(* PLC project BE_Framework BA.project, CODESYS CODESYS V3.5 SP13 Patch 2 *)
(* stored: creationDateTime 2018-12-11T11:00:35.04202, modificationDateTime 2018-12-11T11:00:22.0036737 *)

PROGRAM LB01_FF1_Analog_ST
VAR
	local:strFan_Analog;
	localGP:strSensor2_Regulator;
	ControlFan: _BE_Fan;
	FbRegulator: _BE_Regulator;
	_BE_Fan2: _BE_Fan_2;
	reset_en: RS;
	AlarmFbAl03: _BE_AlarmAckRequired;
	AlarmFbAl02: _BE_AlarmAckRequired;
	fb_OperationalTime: _BE_OperationalTime;
	ackAl01: BOOL;
	ackAl02: BOOL;
	fanGuardOk: BOOL;
END_VAR

            //Struct ->> local
LB01.FF1 := local;
LB01.GP21 := localGP;
LB01.GP23.V := fanGuardOk;

//Fan
IF Local.SP2 > 0 THEN
	local.EnFeedbackError := TRUE;
END_IF

IF Local.SP1 > 0 THEN
	local.EnThermalError := TRUE;
END_IF

IF Local.SP3 > 0 THEN
	local.EnFanGuardError := TRUE;
END_IF

_BE_Fan2.AutoStart := LB01.GeneralStart;
_BE_Fan2.AutoStartTimeDelay := local.SP1 + 5; 
_BE_Fan2.BlockAutoStart := FALSE;
_BE_Fan2.RunIndication := local.V; 
_BE_Fan2.EnableFeedbackAlarm := local.EnFeedbackError; 
_BE_Fan2.FeedbackAlarmTimeDelay := local.SP4; 
_BE_Fan2.EnableThermicRelayAlarm := local.EnThermalError;
_BE_Fan2.ThermicRelayOk := local.ThermoRelay1;
_BE_Fan2.ThermicRelayAlarmTimeDelay := local.SP2;
_BE_Fan2.EnableFanGuardAlarm := local.EnFanGuardError;
_BE_Fan2.FanGuardOk := fanGuardOk;
_BE_Fan2.FanGuardAlarmTimeDelay := local.SP3;
_BE_Fan2.AlarmIndication := local.AL;
_BE_Fan2.AutoReg := local.AUT;

_BE_Fan2();

local.CMD := _BE_Fan2.StartSignalOutput; 
// _BE_Fan2.Status 
local.FeedbackError := _BE_Fan2.FeedbackAlarm;
local.ThermalError := _BE_Fan2.ThermicRelayAlarm;
local.FanGuardError := _BE_Fan2.FanGuardAlarm;

 

//Alarm

//Regulator

//Operational time
fb_OperationalTime(Operating := local.CMD, MinutePulse := SYS_MinutePulse, ResetOperatingTime := local.RST, ResetStarts := local.RST);
local.PV2 := fb_OperationalTime.TotalMinutes;
local.PV1 := fb_OperationalTime.TotalHours;
local.PV3 := fb_OperationalTime.StartsTotal;

//Local --> STRUCT
local := LB01.FF1;
localGP := LB01.GP21;


          
END_PROGRAM
